{attribute addProperty BoxType "EJ1889-0000-0017"}
{attribute addProperty Id "ChannelAT %I*ARRAY[0..15] OF Channel_E4AEF59E128160WcStateAT %I*WcState_F855686C1620InfoDataAT %I*InfoData_192954DE1620"}
{attribute addProperty CRC "3742933219"}
{attribute addProperty SizeInBites "160"}
{attribute addProperty SizeInBytes "20"}
TYPE EJ1889_8059E623 :
STRUCT
	{attribute addProperty Name "Channel"}
	Channel : ARRAY[0..15] OF Channel_E4AEF59E;
	{attribute addProperty Name "WcState"}
	WcState : WcState_F855686C;
	{attribute addProperty Name "InfoData"}
	InfoData : InfoData_192954DE;
END_STRUCT
END_TYPE

(* stored: Version 1.2.0.0, ProductVersion 3.1.4024.9
   DUT EJ1889_8059E623: Id {e75e51c5-f6bf-4add-b30b-b61022d9cc7e} *)
